// TwinCAT 3 PLC project Sample01
// ProgramVersion: 3.1.4020.10
// libraries:
//   Tc2_Standard, * (Beckhoff Automation GmbH)
//   Tc2_System, * (Beckhoff Automation GmbH)
//   Tc3_Module, * (Beckhoff Automation GmbH)
// project tree:
//   / PlcTask.TcTTO (not stored)
//   POUs/ Class Diagram.TcCD (not stored), FB_AnalogValue.TcPOU (not stored), FB_Controller.TcPOU (not stored), FB_Lamp.TcPOU (not stored), FB_LampOnOffAdapter.TcPOU, FB_LampSetDirectAdapter.TcPOU (not stored), FB_LampUpDown.TcPOU, FB_LampSetDirect.TcPOU (not stored), FB_LampOnOff.TcPOU, FB_LampUpDownAdapter.TcPOU (not stored), I_Lamp.TcIO (not stored), I_Observer.TcIO (not stored), I_Subject.TcIO (not stored), MAIN.TcPOU (not stored)
// real-time tasks:
//   TASK PlcTask: cycle T#10ms, priority 20, ADS port 350

// ---- POUs/FB_LampOnOffAdapter.TcPOU
FUNCTION_BLOCK PUBLIC FB_LampOnOffAdapter EXTENDS FB_Lamp
VAR
	fbLampOnOff			: FB_LampOnOff;
END_VAR

// Reduces the control value by 5 in the range of 10 to 100.
METHOD PUBLIC DimDown
fbLampOnOff.DimDown();
IF (_ipObserver <> 0) THEN
	_ipObserver.Update(fbLampOnOff.nLightLevel);
END_IF
END_METHOD

// Increments the control value by 5 in the range of 10 to 100.
METHOD PUBLIC DimUp
fbLampOnOff.DimUp();
IF (_ipObserver <> 0) THEN
	_ipObserver.Update(fbLampOnOff.nLightLevel);
END_IF
END_METHOD

// Sets the control value to 0.
METHOD PUBLIC Off
fbLampOnOff.Off();
IF (_ipObserver <> 0) THEN
	_ipObserver.Update(fbLampOnOff.nLightLevel);
END_IF
END_METHOD

// Sets the control value to 100.
METHOD PUBLIC On
fbLampOnOff.On();
IF (_ipObserver <> 0) THEN
	_ipObserver.Update(fbLampOnOff.nLightLevel);
END_IF
END_METHOD

END_FUNCTION_BLOCK

// ---- POUs/FB_LampOnOff.TcPOU
FUNCTION_BLOCK PUBLIC FB_LampOnOff
VAR
	nLightLevel			: USINT;
END_VAR

// Reduces the control value by 5 in the range of 10 to 100.
METHOD PUBLIC DimDown
Off();
END_METHOD

// Increments the control value by 5 in the range of 10 to 100.
METHOD PUBLIC DimUp
On();
END_METHOD

// Sets the control value to 0.
METHOD PUBLIC Off
nLightLevel := 0;
END_METHOD

// Sets the control value to 100.
METHOD PUBLIC On
nLightLevel := 100;
END_METHOD

END_FUNCTION_BLOCK

// ---- POUs/FB_LampUpDown.TcPOU
FUNCTION_BLOCK FB_LampUpDown
VAR
	nLightLevel			: USINT;
END_VAR

// Reduces the control value by 1 in the range of 10 to 100. 
METHOD PUBLIC OneStepDown
nLightLevel := nLightLevel - 1;
IF (nLightLevel < 10) THEN
	nLightLevel := 10;
END_IF
END_METHOD

// Increments the control value by 1 in the range of 10 to 100.
METHOD PUBLIC OneStepUp
nLightLevel := nLightLevel + 1;
IF (nLightLevel > 100) THEN
	nLightLevel := 100;
END_IF
END_METHOD

// Toggles the control value between 0 and 100.
METHOD PUBLIC OnOff
IF (nLightLevel > 0) THEN
	nLightLevel := 0;
ELSE
	nLightLevel := 100;
END_IF
END_METHOD

END_FUNCTION_BLOCK
